// TIA Portal V17 export
// export: Created 2024-08-07T21:44:12.705008Z, ExportSetting WithDefaults, DisplayName Totally Integrated Automation Portal, DisplayVersion V17 Update 7, DisplayName TIA Portal Openness, DisplayVersion V17 Update 7, DisplayName TIA Portal Version Control Interface, DisplayVersion V17, DisplayName SINAMICS Startdrive Advanced, DisplayVersion V17 SP2, DisplayName SINAMICS Startdrive G110M, G120, G120C, G120D, G120P, G115D, DisplayVersion V17 SP2, DisplayName SINAMICS Startdrive G130, G150, S120, S150, SINAMICS MV, S210, DisplayVersion V17 SP2, DisplayName STEP 7 Professional, DisplayVersion V17 Update 7, DisplayName STEP 7 Safety, DisplayVersion V17 Update 6, DisplayName WinCC Advanced / Unified PC, DisplayVersion V17 Update 7
VAR_GLOBAL   // PLC tag table "Hydraulic"
   iOilTemperature50 AT %I10.0 : Bool;   // cooling only - motor running
   iOilTemperature65 AT %I10.1 : Bool;   // motor stop
   iOilHighLevekOK AT %I10.2 : Bool;
   iOilLowLevelOK AT %I10.3 : Bool;   // stop motor if NOK
   iOilFilter1 AT %I10.4 : Bool;
   iOilFilter2 AT %I10.5 : Bool;
   iOilPressureCupping AT %I10.6 : Bool;
   qHydraulicReductionValveCupforming AT %Q10.1 : Bool;
   aiCupformingLeft AT %IW204 : Int;
   aiCupformingRight AT %IW206 : Int;
   qaCupforming1 AT %QW200 : Int;
   qaCupforming2 AT %QW202 : Int;
   qaReductionCupforming AT %QW204 : Int;
   qHydraulicKM20 AT %Q2.0 : Bool;
   qHydraulicKM21 AT %Q2.1 : Bool;
   iHydraulicCircuitBreakerQ2off AT %I2.4 : Bool;
END_VAR
